{attribute 'GeneratedUsingTerminal: EL5101-0011-0016'}
{attribute addProperty BoxType "EL5101-0011-0016"}
{attribute addProperty Id "StatusAT %I*Status_2E3946CF8"}
{attribute addProperty CRC "1310755001"}
{attribute addProperty Size "8"}
TYPE ENC_Status_4E2088B9 :
STRUCT
	{attribute addProperty Name "Status"}
	Status AT %I* : Status_2E3946CF;
END_STRUCT
END_TYPE

(* stored: Version 1.2.0.0, ProductVersion 3.1.4024.9
   DUT ENC_Status_4E2088B9: Id {854776b2-db45-4278-9542-b684be400189} *)
